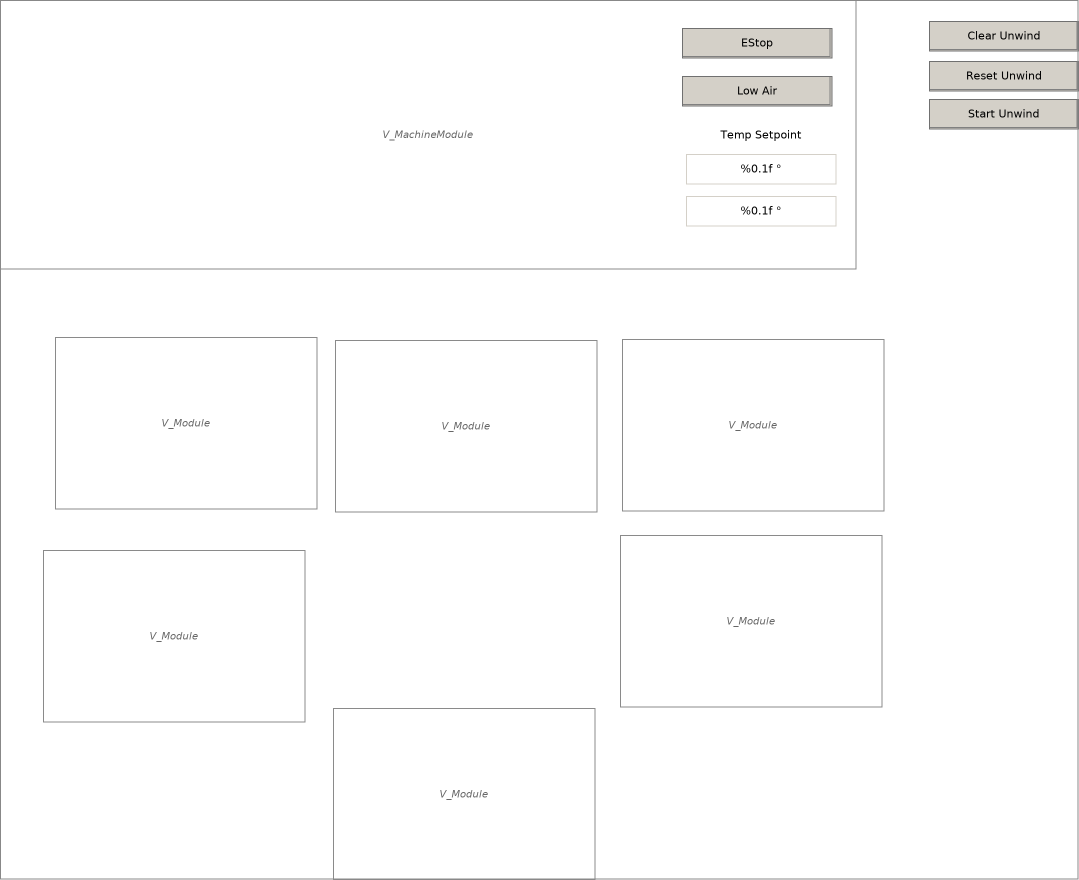
VISUALIZATION V_Main  // 1079x880
    Frame (0,0 856x269)
        shows V_MachineModule(HMI := MAIN.Demo_System.PackMLBaseModule_HMI)
    Frame (43,550 262x172)
        shows V_Module(HMI := MAIN.Demo_System.Station_1.PackMLBaseModule_HMI)
    Frame (55,337 262x172)
        shows V_Module(HMI := MAIN.Demo_System.Station_2.PackMLBaseModule_HMI)
    Frame (335,340 262x172)
        shows V_Module(HMI := MAIN.Demo_System.Station_3.PackMLBaseModule_HMI)
    Button (682,28 150x30), "EStop"
        toggle MAIN.Demo_System.EstopInput
    Button (682,76 150x30), "Low Air"
        toggle MAIN.Demo_System.LowAirInput
    Textfield (686,154 150x30), "%0.1f °", text variable: MAIN.Demo_System.Sealer.SealBar._SetTemperature
        OnMouseDown: write the text variable via VisuDialogs.Numpad, min 20, max 400, title 'Sealer Bar Temp Setpoint', format %0.1f
    Label (686,120 150x30), "Temp Setpoint"
    Textfield (686,196 150x30), "%0.1f °", text variable: MAIN.Demo_System.Sealer.SealBar._ActualTemperature
    Button (929,21 150x30), "Clear Unwind"
        OnMouseClick: execute { MAIN.Demo_System.unwind.PackMLBaseModule_HMI.Command.State := E_PMLCommand.ePMLCommand_Clear; }
    Button (929,61 150x30), "Reset Unwind"
        OnMouseClick: execute { MAIN.Demo_System.unwind.PackMLBaseModule_HMI.Command.State := E_PMLCommand.ePMLCommand_Reset; }
    Button (929,99 150x30), "Start Unwind"
        OnMouseClick: execute { MAIN.Demo_System.unwind.PackMLBaseModule_HMI.Command.State := E_PMLCommand.ePMLCommand_Start; }
    Frame (622,339 262x172)
        shows V_Module(HMI := MAIN.Demo_System.Station_4.PackMLBaseModule_HMI)
    Frame (620,535 262x172)
        shows V_Module(HMI := MAIN.Demo_System.Station_5.PackMLBaseModule_HMI)
    Frame (333,708 262x172)
        shows V_Module(HMI := MAIN.Demo_System.Station_6.PackMLBaseModule_HMI)
END_VISUALIZATION

(* stored: Version 1.1.0.1, ProductVersion 3.1.4024.16
   Visu V_Main: Id {a820fc1e-d71f-479f-a200-f2cc0d18dc0b} *)
